// TIA Portal V15.1 export
// export: Created 2026-01-09T13:45:12.3512035Z, ExportSetting WithDefaults, WithReadOnly, DisplayName Totally Integrated Automation Portal, DisplayVersion V15.1 Update 8, DisplayName TIA Portal Openness, DisplayVersion V15.1 Update 8, DisplayName STEP 7 Professional, DisplayVersion V15.1 Update 8, DisplayName WinCC Advanced, DisplayVersion V15.1 Update 8
FUNCTION "4.CONVERT_VOLUME" : Void   // FC4, LAD
{ S7_Optimized_Access := 'TRUE' }
VERSION : 0.1
// stored: AutoNumber true, CodeModifiedDate 2025-08-27T17:08:03.467369Z, CompileDate 2025-08-30T17:40:35.2171394Z, CreationDate 2024-10-12T12:36:08.0193576Z, HandleErrorsWithinBlock false, InterfaceModifiedDate 2023-07-25T19:47:42.5745Z, IsConsistent true, IsIECCheckEnabled false, IsKnowHowProtected false, IsWriteProtected false, LibraryConformanceStatus The object is library-conformant., ModifiedDate 2025-08-27T17:08:03.467369Z, ParameterModified 2023-07-25T19:47:42.5745Z, PLCSimAdvancedSupport false, SetENOAutomatically False, StructureModified 2023-07-25T19:47:42.5745Z, UDAEnableTagReadback false
   VAR_INPUT
      SO_KHOI : Real;
      M3_MAX : Real;
   END_VAR
   VAR_OUTPUT
      SO_ME : Real;
      "M3/ME" : Real;
   END_VAR
   VAR_TEMP
      TEMP1 : Real;
      TEMP2 : Int;
      TEMP3 : Real;
   END_VAR
BEGIN

REGION Network 1
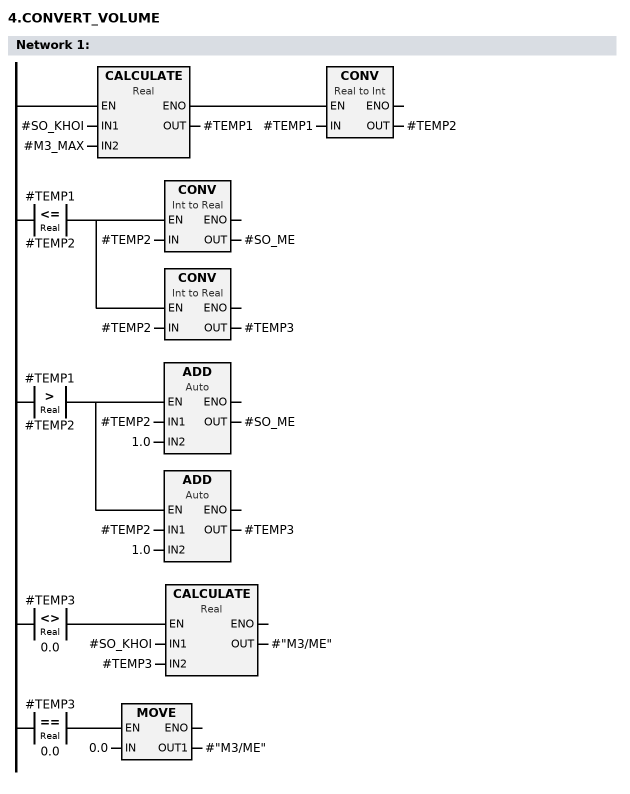
   RUNG wire#powerrail
      { S7_Templates := "SrcType := Real"; S7_Expression := "IN1/IN2" } Calculate(in1 := #SO_KHOI, in2 := #M3_MAX, out => #TEMP1)
      { S7_Templates := "[SrcType := Real, DestType := Int]" } Convert(in := #TEMP1, out => #TEMP2)
   END_RUNG
   RUNG wire#powerrail
      { S7_Templates := "SrcType := Real" } LE_Contact(in1 := #TEMP1, in2 := #TEMP2)
      wire#w1
      { S7_Templates := "[SrcType := Int, DestType := Real]" } Convert(in := #TEMP2, out => #SO_ME)
   END_RUNG
   RUNG wire#w1
      { S7_Templates := "[SrcType := Int, DestType := Real]" } Convert(in := #TEMP2, out => #TEMP3)
   END_RUNG
   RUNG wire#powerrail
      { S7_Templates := "SrcType := Real" } GT_Contact(in1 := #TEMP1, in2 := #TEMP2)
      wire#w2
      Add(in1 := #TEMP2, in2 := 1.0, out => #SO_ME)
   END_RUNG
   RUNG wire#w2
      Add(in1 := #TEMP2, in2 := 1.0, out => #TEMP3)
   END_RUNG
   RUNG wire#powerrail
      { S7_Templates := "SrcType := Real" } NE_Contact(in1 := #TEMP3, in2 := 0.0)
      { S7_Templates := "SrcType := Real"; S7_Expression := "IN1/IN2" } Calculate(in1 := #SO_KHOI, in2 := #TEMP3, out => #"M3/ME")
   END_RUNG
   RUNG wire#powerrail
      { S7_Templates := "SrcType := Real" } EQ_Contact(in1 := #TEMP3, in2 := 0.0)
      Move(in := 0.0, out1 => #"M3/ME")
   END_RUNG
   // the same network as SCL:
   #TEMP1 := #SO_KHOI/#M3_MAX;
   #TEMP2 := REAL_TO_INT(#TEMP1);
   IF #TEMP1 <= #TEMP2 THEN
       #SO_ME := INT_TO_REAL(#TEMP2);
       #TEMP3 := INT_TO_REAL(#TEMP2);
   END_IF;
   IF #TEMP1 > #TEMP2 THEN
       #SO_ME := #TEMP2 + 1.0;
       #TEMP3 := #TEMP2 + 1.0;
   END_IF;
   IF #TEMP3 <> 0.0 THEN #"M3/ME" := #SO_KHOI/#TEMP3; END_IF;
   IF #TEMP3 = 0.0 THEN #"M3/ME" := 0.0; END_IF;
END_REGION
END_FUNCTION
